INTERFACE IACMethodRouteBase EXTENDS IACMethod

METHOD AssignRoute : BOOL
VAR_INPUT
	iAssignWithFunction : IPAProcessFunction;
END_VAR
END_METHOD

PROPERTY FirstCModuleInRoute : IPAControlModule
GET
END_GET
END_PROPERTY

PROPERTY LastCModuleInRoute : IPAControlModule
GET
END_GET
END_PROPERTY

METHOD ResetRoute
VAR_INPUT
END_VAR
END_METHOD

PROPERTY Route : PARoute
GET
END_GET
END_PROPERTY

END_INTERFACE

(* stored: Version 1.1.0.1, ProductVersion 3.1.4020.12
   Itf IACMethodRouteBase: Id {5f0e2e87-cca9-4b49-8d90-0d51c828fc22}
   Method AssignRoute: Id {52a607e6-2781-44dd-9e6a-b3fb46cba777}
   Property FirstCModuleInRoute: Id {eeb4f1ba-7914-48bb-82b7-016bc7aafe51}
   Get Get: Id {50df1f2b-4d94-4022-8af4-373d8a35087d}
   Property LastCModuleInRoute: Id {7744c646-e33a-471d-92a6-002a40ac8936}
   Get Get: Id {9f61e21f-3dc6-4b27-9a1c-b6b357ddfeaa}
   Method ResetRoute: Id {cfbd70f2-7302-48f3-ae05-651a1aefc9f8}
   Property Route: Id {9167d0b2-fd91-43b7-aabc-4dab3ff69b4a}
   Get Get: Id {665e5675-c084-487d-86e4-780b127be625} *)
